Yaskawa INFORM job: 001-R1-HOME.JBI

/JOB
//NAME 001-R1-HOME
//POS
///NPOS 0,0,0,1,0,0
///TOOL 0
///POSTYPE BASE
///RECTAN
///RCONF 1,0,0,0,0,0,0,0,0,0,0,0,0,0,0,0,0,0,0,0,0,0,0,0
P00100=275.000,0.000,875.000,180.0000,45.0000,0.0000
//INST
///DATE 2021/03/25 01:52
///ATTR SC,RW
///GROUP1 RB1
///LVARS 0,1,0,0,0,0,0,0
NOP
' Safe position for R1
MOVJ P100 VJ=10.00
END
